FUNCTION F_GetSubsystemSettings : ST_CFG_Subsystem
(**************************************************************************************
 * 	Application		:	BoxControl Framework
 *	Revision		:	$Revision: 404529 $
 *	Revision date	:	$Date: 2018-04-23 08:21:38 +0200 (Mo., 23 Apr 2018) $
 *	Last changed by	:	$Author: b7bolm $
 *	URL				:	$URL: http://almscdc.swisslog.com/repo/SWPD/Development/BoxControlFramework/20_Release/trunk/01_Software/BCF/BCF/JumpStart/20_Product/10_App/15_Subsystem/10_Lib/10_Conv/10_Functions/F_GetSubSystemSettings.TcPOU $
 *
 *	Purpose			:	Returns group settings
 *
 * ------------------------------------------------------------------------------------
 *	Copyright Swisslog [IP AG], Switzerland. All rights reserved.
 * 
 * ------------------------------------------------------------------------------------
 *	
 * 	Revision History: 
 *
 * 	VERSION			DATE			INITIALS			DESCRIPTION
 *	0.1				01.01.2001		swl					Example
 *
 **************************************************************************************)
VAR
	SubsystemReg	: ST_SubsystemRegistryConv;
END_VAR


// Get Master speed from subsystem
IF __ISVALIDREF(SubsystemRegistry.rSettingsSubsystem) THEN
	// Return Subsystem settings
	F_GetSubsystemSettings := SubsystemRegistry.rSettingsSubsystem;
END_IF

END_FUNCTION

(* stored: Version 1.1.0.1, ProductVersion 3.1.4022.12
   POU F_GetSubSystemSettings: Id {b7a3c98f-4e5c-4b18-8858-4fa1ac80e7eb}, SpecialFunc None *)
